FUNCTION_BLOCK E_RESTART (* Service Interface Function Block Type *)
  (* Standard: 61499-1 Annex A; Description: Copyright (c) 2017 fortiss GmbH This program and the accompanying materials are made available under the terms of the Eclipse Public License 2.0 which is available at https://www.eclipse.org/legal/epl-2.0/ SPDX-License-Identifier: EPL-2.0 *)
  (* Version 1.0, 2017-09-21, Alois Zoitl, fortiss GmbH, initial API and implementation and/or initial documentation *)
  (* Version 3.0, 2025-04-14, Patrick Aigner, changed package *)
  PACKAGE iec61499::events;
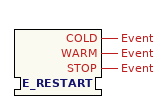
  EVENT_OUTPUT
    COLD; (* Information on cold restart *)
    WARM; (* Information on warm restart *)
    STOP; (* information that the resource is to be stopped *)
  END_EVENT
  SERVICE E_RESTART/RESOURCE (* Service Interface Function Block Type *)
    SEQUENCE cold_restart
      RESOURCE.start() -> E_RESTART.START();
    END_SEQUENCE
    SEQUENCE warm_restart
      RESOURCE.restart() -> E_RESTART.WARM();
    END_SEQUENCE
    SEQUENCE stopping
      RESOURCE.stop() -> E_RESTART.STOP();
    END_SEQUENCE
  END_SERVICE
END_FUNCTION_BLOCK
